FUNCTION_BLOCK FB_MonetPowerMonitoring
VAR_INPUT
END_VAR
VAR_OUTPUT
	phaseOK:				BOOL;
END_VAR
VAR
	fbComm					: I_Comm;	

	// AT%I*/AT%Q* below are mapped directly on this FB: only one instance per PLC is
	// supported, a second instance would collide on the same physical hardware.
	FrequencyGuardWarning	AT%I*: BOOL;
	FrequencyGuardError		AT%I*: BOOL;
	QualityGuardWarning		AT%I*: BOOL;
	QualityGuardError		AT%I*: BOOL;
	UnbalanceGuardWarning	AT%I*: BOOL;
	UnbalanceGuardError		AT%I*: BOOL;
	PowerQuality			AT%I*: REAL;
	L1OverVoltage			AT%I*: BOOL;
	L1InaccVoltage			AT%I*: BOOL;
	L1VoltageGuardWarning	AT%I*: BOOL;
	L1VoltageGuardError		AT%I*: BOOL;
	L2OverVoltage			AT%I*: BOOL;
	L2InaccVoltage			AT%I*: BOOL;
	L2VoltageGuardWarning	AT%I*: BOOL;
	L2VoltageGuardError		AT%I*: BOOL;
	L3OverVoltage			AT%I*: BOOL;
	L3InaccVoltage			AT%I*: BOOL;
	L3VoltageGuardWarning	AT%I*: BOOL;
	L3VoltageGuardError		AT%I*: BOOL;
	
	mqttTimer: 				TON := (PT:=T#10S);
	powerWarningDelay:		TON := (PT:=T#100MS);
	powerWarningRetain:		TOF := (PT:=T#2000MS);
	
	powerError:				FB_EventLog;
	powerWarning:			FB_EventLog;
END_VAR

phaseOK := NOT FrequencyGuardWarning AND NOT L1VoltageGuardWarning AND NOT L2VoltageGuardWarning AND NOT L3VoltageGuardWarning;

powerWarningDelay(IN := NOT phaseOK);
powerWarningRetain(IN := powerWarningDelay.Q);

// MQTT Section
mqttTimer(IN:=TRUE);
IF mqttTimer.Q THEN
	mqttTimer(IN:=FALSE);

	fbComm.Publish('power', 'power', 'FrequencyGuardWarning',	BOOL_TO_STRING(FrequencyGuardWarning));
	fbComm.Publish('power', 'power', 'FrequencyGuardError',	BOOL_TO_STRING(FrequencyGuardError));
	fbComm.Publish('power', 'power', 'QualityGuardWarning',	BOOL_TO_STRING(QualityGuardWarning));
	fbComm.Publish('power', 'power', 'QualityGuardError',		BOOL_TO_STRING(QualityGuardError));
	fbComm.Publish('power', 'power', 'UnbalanceGuardWarning',	BOOL_TO_STRING(UnbalanceGuardWarning));
	fbComm.Publish('power', 'power', 'UnbalanceGuardError',	BOOL_TO_STRING(UnbalanceGuardError));
	fbComm.Publish('power', 'power', 'PowerQuality',			REAL_TO_STRING(PowerQuality));
	fbComm.Publish('power', 'power', 'L1OverVoltage',			BOOL_TO_STRING(L1OverVoltage));
	fbComm.Publish('power', 'power', 'L1InaccVoltage',		BOOL_TO_STRING(L1InaccVoltage));
	fbComm.Publish('power', 'power', 'L1VoltageGuardWarning',	BOOL_TO_STRING(L1VoltageGuardWarning));
	fbComm.Publish('power', 'power', 'L1VoltageGuardError',	BOOL_TO_STRING(L1VoltageGuardError));
	fbComm.Publish('power', 'power', 'L2OverVoltage',			BOOL_TO_STRING(L2OverVoltage));
	fbComm.Publish('power', 'power', 'L2InaccVoltage',		BOOL_TO_STRING(L2InaccVoltage));
	fbComm.Publish('power', 'power', 'L2VoltageGuardWarning',	BOOL_TO_STRING(L2VoltageGuardWarning));
	fbComm.Publish('power', 'power', 'L2VoltageGuardError',	BOOL_TO_STRING(L2VoltageGuardError));
	fbComm.Publish('power', 'power', 'L3OverVoltage',			BOOL_TO_STRING(L3OverVoltage));
	fbComm.Publish('power', 'power', 'L3InaccVoltage',		BOOL_TO_STRING(L3InaccVoltage));
	fbComm.Publish('power', 'power', 'L3VoltageGuardWarning',	BOOL_TO_STRING(L3VoltageGuardWarning));
	fbComm.Publish('power', 'power', 'L3VoltageGuardError',	BOOL_TO_STRING(L3VoltageGuardError));
END_IF

// EventLog section
PowerError(	
	Trigger 		:= FrequencyGuardError OR QualityGuardError OR UnbalanceGuardError OR L1VoltageGuardError OR L2VoltageGuardError OR L3VoltageGuardError, 
	Level 			:= ADSLOG_MSGTYPE_ERROR,
	FormatString 	:= '%s',
	OnMessage 		:= 'electrical power:	ERROR!',
	comm			:= fbComm);
	
PowerWarning(	
	Trigger 		:= powerWarningRetain.Q, 
	Level 			:= ADSLOG_MSGTYPE_WARN,
	FormatString 	:= '%s',
	OnMessage 		:= 'electrical power:	WARNING!',
	comm			:= fbComm);

//FB_Init is always available implicitly and it is used primarily for initialization.
//The return value is not evaluated. For a specific influence, you can also declare the
//methods explicitly and provide additional code there with the standard initialization
//code. You can evaluate the return value.
METHOD FB_Init: BOOL
VAR_INPUT
    bInitRetains	: BOOL; // TRUE: the retain variables are initialized (reset warm / reset cold)
    bInCopyCode		: BOOL;  // TRUE: the instance will be copied to the copy code afterward (online change)
	comm			: I_Comm;	   
END_VAR
THIS^.fbComm := comm;
END_METHOD

END_FUNCTION_BLOCK

(* stored: Version 1.1.0.1, ProductVersion 3.1.4024.15
   POU FB_MonetPowerMonitoring: Id {1c33c5f1-1a01-4451-9e8f-b85db9566c06}, SpecialFunc None
   Method FB_Init: Id {61505fbc-9a86-4110-ab4f-f8109cae6021} *)
